DATA_BLOCK "DB_Robot"
{ S7_Optimized_Access := 'TRUE' }
VERSION : 0.1
NON_RETAIN
"FB_Robot"

BEGIN

END_DATA_BLOCK

